FUNCTION Convert_WORD_TO_DWORD : Hresult
VAR_INPUT
	in : WORD;
	out : REFERENCE TO DWORD;
END_VAR
VAR
	converted : DWORD;
END_VAR

converted := WORD_TO_DWORD(in);

IF (DWORD_TO_WORD(converted) <> in) THEN
	Convert_WORD_TO_DWORD := INCOMPATIBLE;
	RETURN;
END_IF

out := converted;

END_FUNCTION

(* stored: Version 1.1.0.1, ProductVersion 3.1.4024.12
   POU Convert_WORD_TO_DWORD: Id {8abeab5b-2286-48fa-83a6-f8faef367de2}, SpecialFunc None *)
